// TIA Portal V20 export
TYPE "type_emRelations_em8_sequence"
// stored: Access Published, Namespace Unit1
   STRUCT
      hipotThickness : Struct
         jobs : "LAF_typeJobs";
         sequence : "LAF_typeSequence";
         selectJobStatus { S7_SetPoint := 'True'} : Array[0..10] of "LAF_typeJobStatus";
         "step" : "LER_typeStep";
         jobInterface : Struct
            loadJob2 : "LER_typeJobInterface";
            inspectionJob3 : "LER_typeJobInterface";
            unloadJob4 : "LER_typeJobInterface";
         END_STRUCT;
         homeCheck : Struct
            liftDownPartNoDetect : Bool;
            liftDownPartDetect : Bool;
            liftUp : Bool;
         END_STRUCT;
      END_STRUCT;
      hipotThicknessRnR : Struct
         jobs : "LAF_typeJobs";
         sequence : "LAF_typeSequence";
         selectJobStatus { S7_SetPoint := 'True'} : Array[0..10] of "LAF_typeJobStatus";
         "step" : "LER_typeStep";
         jobInterface : Struct
            loadJob2 : "LER_typeJobInterface";
            inspectionJob3 : "LER_typeJobInterface";
            unloadJob4 { S7_SetPoint := 'True'} : "LER_typeJobInterface";
         END_STRUCT;
      END_STRUCT;
   END_STRUCT;
   // // hipotThickness."step".action1[101] : Step[101] : JOB[1] Condition
   // // hipotThickness."step".action1[110] : Step[110] : Hipot & Thickness Z-Axis Wait Pos
   // // hipotThickness."step".action1[111] : Step[111] : Servo Press Reference Home Pos
   // // hipotThickness."step".action1[120] : Step[120] : Tab Contactor Open
   // // hipotThickness."step".action1[121] : Step[121] : Tab Contactor Backward
   // // hipotThickness."step".action1[130] : Step[130] : Stage Lift Up
   // // hipotThickness."step".action1[140] : Step[140] : Spare
   // // hipotThickness."step".action1[150] : Step[150] : Stage Lift Down
   // // hipotThickness."step".action1[170] : Step[170] : Spare
   // // hipotThickness."step".action1[190] : Step[190] : JOB[1] Step End
   // // hipotThickness."step".action1[201] : Step[201] : JOB[2] Condition
   // // hipotThickness."step".action1[210] : Step[210] : Hipot & Thickness Loading Request => Transfer PP Left
   // // hipotThickness."step".action1[220] : Step[220] : Spare
   // // hipotThickness."step".action1[230] : Step[230] : Stage Lift Up
   // // hipotThickness."step".action1[240] : Step[240] : Hipot & Thickness Loading Check => Transfer PP Left
   // // hipotThickness."step".action1[250] : Step[250] : Spare
   // // hipotThickness."step".action1[290] : Step[290] : JOB[2] Step End
   // // hipotThickness."step".action1[301] : Step[301] : JOB[3] Condition
   // // hipotThickness."step".action1[310] : Step[310] : Stage Lift Down
   // // hipotThickness."step".action1[311] : Step[311] : Stage JR Detection Check
   // // hipotThickness."step".action1[320] : Step[320] : Spare
   // // hipotThickness."step".action1[330] : Step[330] : Press Start
   // // hipotThickness."step".action1[331] : Step[331] : Press Result
   // // hipotThickness."step".action1[340] : Step[340] : Thickness Z-Axis Thickness Ready Pos, Tab Forward
   // // hipotThickness."step".action1[341] : Step[341] : Thickness Z-Axis Measuring Thickness Pos, Tab Contactor Close
   // // hipotThickness."step".action1[350] : Step[350] : Thickness Start
   // // hipotThickness."step".action1[351] : Step[351] : Thickness Result
   // // hipotThickness."step".action1[352] : Step[352] : Thickness Z-Axis Wait Pos
   // // hipotThickness."step".action1[360] : Step[360] : Hipot Start
   // // hipotThickness."step".action1[361] : Step[361] : Hipot Result
   // // hipotThickness."step".action1[362] : Step[362] : Tab Contactor Open
   // // hipotThickness."step".action1[363] : Step[363] : Tab Contactor Backward
   // // hipotThickness."step".action1[380] : Step[380] : Press Home
   // // hipotThickness."step".action1[390] : Step[390] : JOB[3] Step End
   // // hipotThickness."step".action1[401] : Step[401] : JOB[4] Condition
   // // hipotThickness."step".action1[410] : Step[410] : Spare
   // // hipotThickness."step".action1[420] : Step[420] : Stage Lift Up
   // // hipotThickness."step".action1[430] : Step[430] : Hipot & Thickness Unloading Request => Transfer PP Right
   // // hipotThickness."step".action1[431] : Step[431] : Hipot & Thickness Unloading Check => Transfer PP Right
   // // hipotThickness."step".action1[480] : Step[480] : Stage Lift Down
   // // hipotThickness."step".action1[481] : Step[481] : Spare
   // // hipotThickness."step".action1[490] : Step[490] : JOB[4] Step End
   // // hipotThickness."step".transition1[101] : Step[101] : JOB[1] Condition
   // // hipotThickness."step".transition1[110] : Step[110] : Hipot & Thickness Z-Axis Wait Pos
   // // hipotThickness."step".transition1[111] : Step[111] : Servo Press Reference Home Pos
   // // hipotThickness."step".transition1[120] : Step[120] : Tab Contactor Open
   // // hipotThickness."step".transition1[121] : Step[121] : Tab Contactor Backward
   // // hipotThickness."step".transition1[130] : Step[130] : Stage Lift Up
   // // hipotThickness."step".transition1[140] : Step[140] : Spare
   // // hipotThickness."step".transition1[150] : Step[150] : Stage Lift Down
   // // hipotThickness."step".transition1[170] : Step[170] : Spare
   // // hipotThickness."step".transition1[190] : Step[190] : JOB[1] Step End
   // // hipotThickness."step".transition1[201] : Step[201] : JOB[2] Condition
   // // hipotThickness."step".transition1[210] : Step[210] : Hipot & Thickness Loading Request => Transfer PP Left
   // // hipotThickness."step".transition1[220] : Step[220] : Spare
   // // hipotThickness."step".transition1[230] : Step[230] : Stage Lift Up
   // // hipotThickness."step".transition1[240] : Step[240] : Hipot & Thickness Loading Check => Transfer PP Left
   // // hipotThickness."step".transition1[250] : Step[250] : Spare
   // // hipotThickness."step".transition1[290] : Step[290] : JOB[2] Step End
   // // hipotThickness."step".transition1[301] : Step[301] : JOB[3] Condition
   // // hipotThickness."step".transition1[310] : Step[310] : Stage Lift Down
   // // hipotThickness."step".transition1[311] : Step[311] : Stage JR Detection Check
   // // hipotThickness."step".transition1[320] : Step[320] : Spare
   // // hipotThickness."step".transition1[330] : Step[330] : Press Start
   // // hipotThickness."step".transition1[331] : Step[331] : Press Result
   // // hipotThickness."step".transition1[340] : Step[340] : Thickness Z-Axis Thickness Ready Pos, Tab Forward
   // // hipotThickness."step".transition1[341] : Step[341] : Thickness Z-Axis Measuring Thickness Pos, Tab Contactor Close
   // // hipotThickness."step".transition1[350] : Step[350] : Thickness Start
   // // hipotThickness."step".transition1[351] : Step[351] : Thickness Result
   // // hipotThickness."step".transition1[352] : Step[352] : Thickness Z-Axis Wait Pos
   // // hipotThickness."step".transition1[360] : Step[360] : Hipot Start
   // // hipotThickness."step".transition1[361] : Step[361] : Hipot Result
   // // hipotThickness."step".transition1[362] : Step[362] : Tab Contactor Open
   // // hipotThickness."step".transition1[363] : Step[363] : Tab Contactor Backward
   // // hipotThickness."step".transition1[380] : Step[380] : Press Home
   // // hipotThickness."step".transition1[390] : Step[390] : JOB[3] Step End
   // // hipotThickness."step".transition1[401] : Step[401] : JOB[4] Condition
   // // hipotThickness."step".transition1[410] : Step[410] : Spare
   // // hipotThickness."step".transition1[420] : Step[420] : Stage Lift Up
   // // hipotThickness."step".transition1[430] : Step[430] : Hipot & Thickness Unloading Request => Transfer PP Right
   // // hipotThickness."step".transition1[431] : Step[431] : Hipot & Thickness Unloading Check => Transfer PP Right
   // // hipotThickness."step".transition1[480] : Step[480] : Stage Lift Down
   // // hipotThickness."step".transition1[481] : Step[481] : Spare
   // // hipotThickness."step".transition1[490] : Step[490] : JOB[4] Step End
   // // hipotThicknessRnR."step".action1[101] : Step[101] : JOB[1] Condition
   // // hipotThicknessRnR."step".action1[110] : Step[110] : Hipot & Thickness Z-Axis Wait Pos
   // // hipotThicknessRnR."step".action1[111] : Step[111] : Servo Press Reference Home Pos
   // // hipotThicknessRnR."step".action1[120] : Step[120] : Tab Contactor Open
   // // hipotThicknessRnR."step".action1[121] : Step[121] : Tab Contactor Backward
   // // hipotThicknessRnR."step".action1[130] : Step[130] : Stage Lift Up
   // // hipotThicknessRnR."step".action1[140] : Step[140] : Spare
   // // hipotThicknessRnR."step".action1[150] : Step[150] : Stage Lift Down
   // // hipotThicknessRnR."step".action1[170] : Step[170] : Spare
   // // hipotThicknessRnR."step".action1[190] : Step[190] : JOB[1] Step End
   // // hipotThicknessRnR."step".action1[201] : Step[201] : JOB[2] Condition
   // // hipotThicknessRnR."step".action1[210] : Step[210] : Hipot & Thickness Loading Request => Transfer PP Left
   // // hipotThicknessRnR."step".action1[220] : Step[220] : Spare
   // // hipotThicknessRnR."step".action1[230] : Step[230] : Stage Lift Up
   // // hipotThicknessRnR."step".action1[240] : Step[240] : Hipot & Thickness Loading Check => Transfer PP Left
   // // hipotThicknessRnR."step".action1[250] : Step[250] : Spare
   // // hipotThicknessRnR."step".action1[290] : Step[290] : JOB[2] Step End
   // // hipotThicknessRnR."step".action1[301] : Step[301] : JOB[3] Condition
   // // hipotThicknessRnR."step".action1[310] : Step[310] : Stage Lift Down
   // // hipotThicknessRnR."step".action1[311] : Step[311] : Stage JR Detection Check
   // // hipotThicknessRnR."step".action1[320] : Step[320] : Spare
   // // hipotThicknessRnR."step".action1[330] : Step[330] : Press Start
   // // hipotThicknessRnR."step".action1[331] : Step[331] : Press Result
   // // hipotThicknessRnR."step".action1[340] : Step[340] : Thickness Z-Axis Thickness Ready Pos, Tab Forward
   // // hipotThicknessRnR."step".action1[341] : Step[341] : Thickness Z-Axis Measuring Thickness Pos, Tab Contactor Close
   // // hipotThicknessRnR."step".action1[350] : Step[350] : Thickness Start
   // // hipotThicknessRnR."step".action1[351] : Step[351] : Thickness Result
   // // hipotThicknessRnR."step".action1[352] : Step[352] : Thickness Z-Axis Wait Pos
   // // hipotThicknessRnR."step".action1[360] : Step[360] : Hipot Start
   // // hipotThicknessRnR."step".action1[361] : Step[361] : Hipot Result
   // // hipotThicknessRnR."step".action1[362] : Step[362] : Tab Contactor Open
   // // hipotThicknessRnR."step".action1[363] : Step[363] : Tab Contactor Backward
   // // hipotThicknessRnR."step".action1[380] : Step[380] : Press Home
   // // hipotThicknessRnR."step".action1[390] : Step[390] : JOB[3] Step End
   // // hipotThicknessRnR."step".action1[401] : Step[401] : JOB[4] Condition
   // // hipotThicknessRnR."step".action1[410] : Step[410] : Spare
   // // hipotThicknessRnR."step".action1[420] : Step[420] : Stage Lift Up
   // // hipotThicknessRnR."step".action1[430] : Step[430] : Hipot & Thickness Unloading Request => Transfer PP Right
   // // hipotThicknessRnR."step".action1[431] : Step[431] : Hipot & Thickness Unloading Check => Transfer PP Right
   // // hipotThicknessRnR."step".action1[480] : Step[480] : Stage Lift Down
   // // hipotThicknessRnR."step".action1[481] : Step[481] : Spare
   // // hipotThicknessRnR."step".action1[490] : Step[490] : JOB[4] Step End
   // // hipotThicknessRnR."step".transition1[101] : Step[101] : JOB[1] Condition
   // // hipotThicknessRnR."step".transition1[110] : Step[110] : Hipot & Thickness Z-Axis Wait Pos
   // // hipotThicknessRnR."step".transition1[111] : Step[111] : Servo Press Reference Home Pos
   // // hipotThicknessRnR."step".transition1[120] : Step[120] : Tab Contactor Open
   // // hipotThicknessRnR."step".transition1[121] : Step[121] : Tab Contactor Backward
   // // hipotThicknessRnR."step".transition1[130] : Step[130] : Stage Lift Up
   // // hipotThicknessRnR."step".transition1[140] : Step[140] : Spare
   // // hipotThicknessRnR."step".transition1[150] : Step[150] : Stage Lift Down
   // // hipotThicknessRnR."step".transition1[170] : Step[170] : Spare
   // // hipotThicknessRnR."step".transition1[190] : Step[190] : JOB[1] Step End
   // // hipotThicknessRnR."step".transition1[201] : Step[201] : JOB[2] Condition
   // // hipotThicknessRnR."step".transition1[210] : Step[210] : Hipot & Thickness Loading Request => Transfer PP Left
   // // hipotThicknessRnR."step".transition1[220] : Step[220] : Spare
   // // hipotThicknessRnR."step".transition1[230] : Step[230] : Stage Lift Up
   // // hipotThicknessRnR."step".transition1[240] : Step[240] : Hipot & Thickness Loading Check => Transfer PP Left
   // // hipotThicknessRnR."step".transition1[250] : Step[250] : Spare
   // // hipotThicknessRnR."step".transition1[290] : Step[290] : JOB[2] Step End
   // // hipotThicknessRnR."step".transition1[301] : Step[301] : JOB[3] Condition
   // // hipotThicknessRnR."step".transition1[310] : Step[310] : Stage Lift Down
   // // hipotThicknessRnR."step".transition1[311] : Step[311] : Stage JR Detection Check
   // // hipotThicknessRnR."step".transition1[320] : Step[320] : Spare
   // // hipotThicknessRnR."step".transition1[330] : Step[330] : Press Start
   // // hipotThicknessRnR."step".transition1[331] : Step[331] : Press Result
   // // hipotThicknessRnR."step".transition1[340] : Step[340] : Thickness Z-Axis Thickness Ready Pos, Tab Forward
   // // hipotThicknessRnR."step".transition1[341] : Step[341] : Thickness Z-Axis Measuring Thickness Pos, Tab Contactor Close
   // // hipotThicknessRnR."step".transition1[350] : Step[350] : Thickness Start
   // // hipotThicknessRnR."step".transition1[351] : Step[351] : Thickness Result
   // // hipotThicknessRnR."step".transition1[352] : Step[352] : Thickness Z-Axis Wait Pos
   // // hipotThicknessRnR."step".transition1[360] : Step[360] : Hipot Start
   // // hipotThicknessRnR."step".transition1[361] : Step[361] : Hipot Result
   // // hipotThicknessRnR."step".transition1[362] : Step[362] : Tab Contactor Open
   // // hipotThicknessRnR."step".transition1[363] : Step[363] : Tab Contactor Backward
   // // hipotThicknessRnR."step".transition1[380] : Step[380] : Press Home
   // // hipotThicknessRnR."step".transition1[390] : Step[390] : JOB[3] Step End
   // // hipotThicknessRnR."step".transition1[401] : Step[401] : JOB[4] Condition
   // // hipotThicknessRnR."step".transition1[410] : Step[410] : Spare
   // // hipotThicknessRnR."step".transition1[420] : Step[420] : Stage Lift Up
   // // hipotThicknessRnR."step".transition1[430] : Step[430] : Hipot & Thickness Unloading Request => Transfer PP Right
   // // hipotThicknessRnR."step".transition1[431] : Step[431] : Hipot & Thickness Unloading Check => Transfer PP Right
   // // hipotThicknessRnR."step".transition1[480] : Step[480] : Stage Lift Down
   // // hipotThicknessRnR."step".transition1[481] : Step[481] : Spare
   // // hipotThicknessRnR."step".transition1[490] : Step[490] : JOB[4] Step End
END_TYPE
